FUNCTION POU : BOOL
VAR_INPUT
END_VAR
VAR
END_VAR

END_FUNCTION

(* stored: Version 1.1.0.1, ProductVersion 3.1.4024.12
   POU POU: Id {73589837-d2c9-40a7-9aee-c76a33b51521}, SpecialFunc None *)
